// TIA Portal V16 export
// export: Created 2021-07-12T14:47:18.4124345Z, ExportSetting WithDefaults, DisplayName Totally Integrated Automation Portal, DisplayVersion V16, DisplayName TIA Portal Version Control Interface, DisplayVersion V16, DisplayName TIA Portal Openness, DisplayVersion V16, DisplayName STEP 7 Professional, DisplayVersion V16, DisplayName STEP 7 Safety, DisplayVersion V16, DisplayName WinCC Professional, DisplayVersion V16
TYPE "LSimaHydTO_typeInternalStatusDirectOutput"
TITLE = LSimaHydTO_typeInternalStatusDirectOutput
// Manual output control
// stored: IsFailsafeCompliant false
   STRUCT
      active : Bool;   // displays activity of manual output operation
      rampingDown : Bool;   // ramping down due to positioning limits
      minSafetyPositionOverrun : Bool;   // the min. safety position was passed
      maxSafetyPositionOverrun : Bool;   // the max. safety position was passed
      QOutputValue : LReal;
      cmdTracking { S7_SetPoint := 'True'} : "LSimaHydTO_typeInternalCmdTracking";
   END_STRUCT;
END_TYPE
